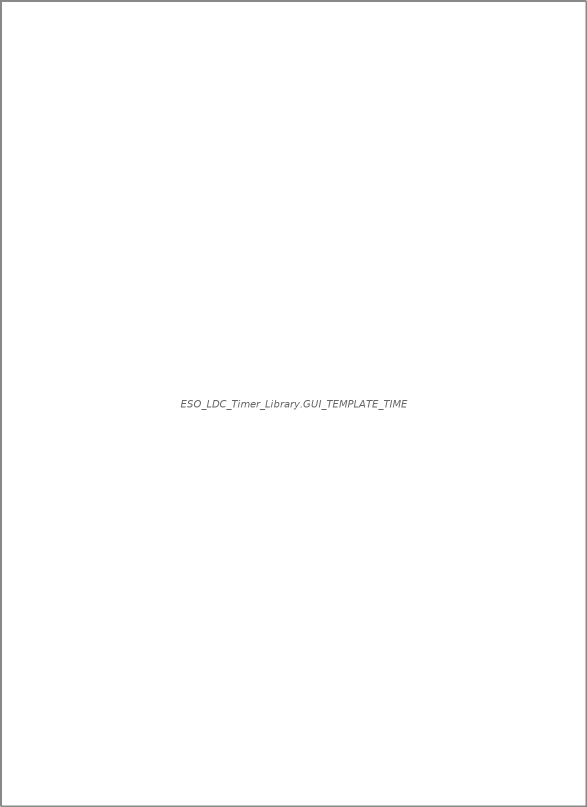
VISUALIZATION GUI_TIME_INFORMATION  // 587x807
    Frame (1,1 586x806)
        shows ESO_LDC_Timer_Library.GUI_TEMPLATE_TIME(m_Instance := MAIN.time_info)
END_VISUALIZATION

(* stored: Version 1.1.0.1, ProductVersion 3.1.4024.12
   Visu GUI_TIME_INFORMATION: Id {8d096512-7dcb-478d-be90-e286b18e5747} *)
